FUNCTION ScalingIn : BOOL
VAR_INPUT
END_VAR
VAR
END_VAR

Process.currentHeight:= Inputs.AI_HEIGHT*(0.0263) + 79.878;
IIRFilter(Process.currentHeight,0.99,Process.Height);
//Process.Height := Inputs.AI_HEIGHT*(-0.00508825) + 49.10937731;

// Circulation system pressure
Process.Pressure := Inputs.AI_PressureSensor*0.003277 - 0.12124;

// Circluation system temperature
Process.Temperature := Inputs.AI_TEMP*0.003282 - 0.1083;

END_FUNCTION

(* stored: Version 1.1.0.1, ProductVersion 3.1.4024.9
   POU ScalingIn: Id {a75abb54-6290-4759-8cf7-84d3613d9788}, SpecialFunc None *)
